KUKA KRL data list: cleanup.dat

&ACCESS RV1
DEFDAT  cleanup PUBLIC

ENDDAT
